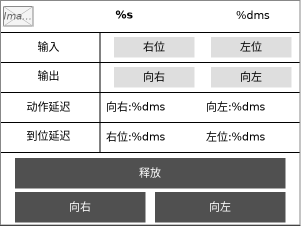
VISUALIZATION Cyliner4  // 301x226
VAR_INPUT
	System:							REFERENCE TO ST_System;
	Cylinder:						REFERENCE TO ST_Cylinder;
	CylinderData:					REFERENCE TO ST_CylinderData;
END_VAR
    RoundedRectangle (0,111 300x115)
    RoundedRectangle (0,0 300x115)
    Rectangle (0,34 300x115)
    Line (0,32) (300,32)
    Rectangle (35,3 179x24), "%s", text variable: Cylinder.arrInfo[System.stMode.eLanguage].sName, input disabled if: Cylinder.stLock.bShield
    Rectangle (218,3 70x25), "%dms", text variable: CylinderData.iAlarmTime, input disabled if: Cylinder.stLock.bShield
        OnMouseClick: write the text variable via VisuDialogs.Numpad
    Line (0,62) (300,62)
    Line (0,92) (300,92)
    Label (1,32 95x30), "输入"
    Label (1,61 95x30), "输出"
    Line (100,152) (100,32)
    RoundedRectangle (114,37 80x20), "右位", colour toggle: Cylinder.stInput.bWork, input disabled if: Cylinder.stLock.bShield
    RoundedRectangle (211,37 80x20), "左位", colour toggle: Cylinder.stInput.bHome, input disabled if: Cylinder.stLock.bShield
    RoundedRectangle (114,67 80x20), "向右", colour toggle: Cylinder.stOutput.bWork, input disabled if: Cylinder.stLock.bShield
    RoundedRectangle (211,67 80x20), "向左", colour toggle: Cylinder.stOutput.bHome, input disabled if: Cylinder.stLock.bShield
    RoundedRectangle (15,158 270x30), "释放", colour toggle: Cylinder.stLock.bOff OR Cylinder.stLock.bAll, input disabled if: Cylinder.stLock.bShield
        tap Cylinder.stControl.stOffRequest.bManual
    RoundedRectangle (15,192 130x30), "向右", colour toggle: Cylinder.stLock.bWork OR Cylinder.stLock.bAll, input disabled if: Cylinder.stLock.bShield
        tap Cylinder.stControl.stWorkRequest.bManual
    RoundedRectangle (155,192 130x30), "向左", colour toggle: Cylinder.stLock.bHome OR Cylinder.stLock.bAll, input disabled if: Cylinder.stLock.bShield
        tap Cylinder.stControl.stHomeRequest.bManual
    Line (300,154) (300,23)
    Line (0,152) (0,19)
    Image (3,6 30x20), image: ImagePool.Cylinder1
    Line (0,122) (300,122)
    Line (0,152) (300,152)
    Label (1,92 95x30), "动作延迟"
    Label (1,121 95x30), "到位延迟"
    RoundedRectangle (103,94 95x26), "向右:%dms", text variable: CylinderData.iWorkRequestTime, input disabled if: Cylinder.stLock.bShield
        OnMouseClick: write the text variable via Default
    RoundedRectangle (203,94 95x26), "向左:%dms", text variable: CylinderData.iHomeRequestTime, input disabled if: Cylinder.stLock.bShield
        OnMouseClick: write the text variable via Default
    RoundedRectangle (103,124 95x26), "右位:%dms", text variable: CylinderData.iWorkDone, input disabled if: Cylinder.stLock.bShield
        OnMouseClick: write the text variable via Default
    RoundedRectangle (203,124 95x26), "左位:%dms", text variable: CylinderData.iHomeDone, input disabled if: Cylinder.stLock.bShield
        OnMouseClick: write the text variable via Default
END_VISUALIZATION

(* stored: Version 1.1.0.1, ProductVersion 3.1.4024.4
   Visu Cyliner4: Id {fbff16c9-411c-438d-bbdc-7358ff1a7100} *)
